(* LS Electric XG5000 project: Test_260202 *)
(* PLC LSPLC *)
(* module base 0 slot 0: FEnet:XGL-EFMT(B) (Fast Ethernet 통신 모듈, 전기 Master) *)
(* module base 0 slot 1: 입력 모듈:XGI-D21A (DC 24V 입력, 8점 (전류소스/싱크입력)) *)
(* module base 0 slot 2: 출력 모듈:XGQ-RY1A (릴레이 출력, 8점 (2A용, 단독 COM.)) *)

(* Comments on direct variables
%MX0	Emitter 0 (Emit)
%MX1	E_Belt 0
%MX2	Emitter 1 (Emit)
%MX3	E_Belt 1
%MX4	Emitter 2 (Emit)
%MX5	E_Belt 2
%MX6	Emitter 3 (Emit)
%MX7	E_Belt 3
%MX8	Emitter 4 (Emit)
%MX9	E_Belt 4
%MX10	Emitter 5 (Emit)
%MX11	E_Belt 5
%MX12	P_Belt00
%MX13	Sensor P_Belt00_E
%MX14	P_Belt0
%MX15	Sensor P_Belt0_E
%MX16	Sensor P_Belt0_S
%MX17	P_Belt1
%MX18	Sensor P_Belt1_E
%MX19	Sensor P_Belt1_S
%MX20	P_Belt2
%MX21	Sensor P_Belt2_E
%MX22	Sensor P_Belt2_S
%MX23	P_Belt3
%MX24	Sensor P_Belt3_E
%MX25	Sensor P_Belt3_S
%MX26	P_Belt4
%MX27	Sensor P_Belt4_E
%MX28	Sensor P_Belt4_S
%MX29	P_Belt5
%MX30	Sensor P_Belt5_E
%MX31	Sensor P_Belt5_S
%MX32	P_Belt6
%MX33	Sensor P_Belt6_S
%MX34	Sensor P_Belt6_E
%MX35	CC_Belt0
%MX36	Sensor CC_Belt0
%MX37	Sensor CC_Belt1
%MX38	Sensor CC_Belt2
%MX39	Pusher 0
%MX40	Pusher 1
%MX41	Pusher 2
%MX42	Pusher 3
%MX43	Pusher 4
%MX44	CG_Belt1
%MX45	CG_Belt2
%MX46	CG_Curved Belt0
%MX47	CGD_Belt0
%MX48	CGD_Belt1
%MX49	CGD_Belt2
%MX50	CGD_Belt3
%MX51	Sensor Divide_G
%MX52	Sensor Error0
%MX53	Sensor_Count_Green
%MX54	CB_Belt1
%MX55	CB_Curved Belt0
%MX56	CBD_Belt0
%MX57	CBD_Belt1
%MX58	CBD_Belt2
%MX59	CBD_Belt3
%MX60	CBD_Belt4
%MX61	Pusher 5
%MX62	Pusher 6
%MX63	Sensor Divide_B
%MX64	Sensor Error1
%MX65	Sensor_Count_Blue
%MX66	CM_Belt1
%MX67	CM_Curved Belt0
%MX68	CMD_Belt0
%MX69	CMD_Belt1
%MX70	CMD_Belt2
%MX71	CMD_Belt3
%MX72	CMD_Belt4
%MX73	Pusher 7
%MX74	Pusher 8
%MX75	Sensor Divide_M
%MX76	Sensor Error2
%MX77	Sensor_Count_Metal
%MX100	A_Belt blue Conveyor
%MX101	A_Entry conveyor
%MX102	A_Start Entry Conveyor
%MX103	A_Item at entry
%MX104	A_Box at place
%MX105	A_Box Pass
%MX106	A_Box exit Conveyor
%MX107	A_Chain Transfer1 
%MX108	A_Chain Transfer2
%MX109	A_Transfer1 (Left)
%MX110	A_Transfer2 (Left)
%MX111	A_Direction Change
%MX112	A_Box entry to ware
%MX113	A_Box entry warehouse
%MX114	A_Box Check
%MX115	WA_Entry conveyor
%MX116	B_Belt Green Conveyor
%MX117	B_Entry conveyor
%MX118	B_Start Entry Conveyor
%MX119	B_Item at entry
%MX120	B_Box at place
%MX121	B_Box Pass
%MX122	B_Box exit Conveyor1
%MX123	B_Go
%MX124	B_Box arrive
%MX125	B_return
%MX126	B_Box Pass2
%MX127	B_Box exit Conveyor2
%MX128	B_Chain Transfer1 
%MX129	B_Chain Transfer2
%MX130	B_Direction Change
%MX131	B_Transfer1 (Right)
%MX132	B_Transfer2 (Right)
%MX133	B_Box entry to ware
%MX134	B_Box entry warehouse
%MX135	B_Box Check
%MX136	WB_Entry conveyor
%MX137	C_Belt Gray Conveyor
%MX138	C_Start Entry Conveyor
%MX139	C_Entry conveyor
%MX140	C_Item at entry
%MX141	C_Exit Conveyor
%MX142	C_Box Pass
%MX143	C_Box Pass2
%MX144	C_Exit Conveyor
%MX145	C_Chain Transfer1 
%MX146	C_Chain Transfer2
%MX147	C_Direction Change
%MX148	C_Transfer1 (Right)
%MX149	C_Transfer2 (Right)
%MX150	C_Box entry to ware
%MX151	C_Box entry warehouse
%MX152	WC_Entry conveyor
%MX500	Out_Conv_1_In_Sensor
%MX501	Out_Conv_1_Out_Sensor
%MX502	Out_Conv_2_In_Sensor
%MX503	Out_Conv_2_Out_Sensor
%MX504	Out_Conv_3_In_Sensor
%MX505	Out_Conv_3_Out_Sensor
%MX506	Out_Conv_4_In_Sensor
%MX507	Out_Conv_4_Out_Sensor
%MX508	Out_Conv_Line1-1_In_Sensor
%MX509	Out_Conv_Line1-1_Out_Sensor
%MX510	Out_Conv_Line1-2_In_Sensor
%MX511	Out_Conv_Line1-2_Out_Sensor
%MX512	Out_Conv_Line1-3_In_Sensor
%MX513	Out_Conv_Line1-3_Out_Sensor
%MX514	Out_Conv_Line1-4_In_Sensor
%MX515	Out_Conv_Line1-4_Out_Sensor
%MX516	Out_Conv_Line2-1_In_Sensor
%MX517	Out_Conv_Line2-1_Out_Sensor
%MX518	Out_Conv_Line2-2_In_Sensor
%MX519	Out_Conv_Line2-2_Out_Sensor
%MX520	Out_Conv_Line2-3_In_Sensor
%MX521	Out_Conv_Line2-3_Out_Sensor
%MX522	Out_Conv_Line2-4_In_Sensor
%MX523	Out_Conv_Line2-4_Out_Sensor
%MX524	Out_Conv_Line2-5_In_Sensor
%MX525	Out_Conv_Line2-5_Out_Sensor
%MX526	Out_Conv_Line3-1_In_Sensor
%MX527	Out_Conv_Line3-1_Out_Sensor
%MX528	Out_Conv_Line3-2_In_Sensor
%MX529	Out_Conv_Line3-2_Out_Sensor
%MX530	Out_Conv_Line3-3_In_Sensor
%MX531	Out_Conv_Line3-3_Out_Sensor
%MX532	Out_Conv_Line3-4_In_Sensor
%MX533	Out_Conv_Line3-4_Out_Sensor
%MX1000	Start_Button 0
%MX1001	Stop_Button 0
%MX1002	Emergency Stop 0
%MX1003	Machining Center 0 (Is Busy)
%MX1004	Machining Center 0 (Has Error)
%MX1005	Start_Button 1
%MX1006	Stop_Button 1
%MX1007	Emergency Stop 1
%MX1008	Machining Center 1 (Is Busy)
%MX1009	Machining Center 1 (Has Error)
%MX1010	Start_Button 2
%MX1011	Stop_Button 2
%MX1012	Emergency Stop 2
%MX1013	Machining Center 2 (Is Busy)
%MX1014	Machining Center 2 (Has Error)
%MX1015	Start_Button 3
%MX1016	Stop_Button 3
%MX1017	Emergency Stop 3
%MX1018	Machining Center 3 (Is Busy)
%MX1019	Machining Center 3 (Has Error)
%MX1020	C_Start Button 0
%MX1021	C_Stop Button 0
%MX1022	C_Emergency Stop 0
%MX1023	Vision Sensor 0
%MX1024	Vision Sensor 1
%MX1025	Vision Sensor 2
%MX1026	Vision Sensor 3
%MX1027	Vision Sensor 4
%MX1028	Vision Sensor 5
%MX1029	Pusher 0 (Front Limit)
%MX1030	Pusher 1 (Front Limit)
%MX1031	Pusher 2 (Front Limit)
%MX1032	Vision Sensor 6
%MX1033	Vision Sensor 7
%MX1034	Vision Sensor 8
%MX1035	Vision Sensor 9
%MX1036	Vision Sensor 10
%MX1037	Vision Sensor 11
%MX1038	Pusher 3 (Front Limit)
%MX1039	Pusher 4 (Front Limit)
%MX1040	Pusher 5 (Front Limit)
%MX1041	Pusher 6 (Front Limit)
%MX1042	Pusher 7 (Front Limit)
%MX1043	Pusher 8 (Front Limit)
%MX1044	Diffuse Sensor 4
%MX1045	Diffuse Sensor 5
%MX1046	Right Positioner 0 (Clamped)
%MX1047	Right Positioner 1 (Clamped)
%MX1048	Two-Axis Pick & Place 0 (Detected)
%MX1049	Two-Axis Pick & Place 0 (Moving X)
%MX1050	Two-Axis Pick & Place 0 (Moving Z)
%MX1051	Clamp_Sensor 0
%MX1052	Clamp_Sensor 1
%MX1053	Combine Sensor 0
%MX1054	RaiseDown_Sensor 0
%MX1055	Start_Button 4
%MX1056	Stop_Button 4
%MX1057	Emergency Stop 4
%MX1058	Machining Center 4 (Is Busy)
%MX1059	Machining Center 4 (Has Error)
%MX1060	Start_Button 5
%MX1061	Stop_Button 5
%MX1062	Emergency Stop 5
%MX1063	Machining Center 5 (Is Busy)
%MX1064	Machining Center 5 (Has Error)
%MX1065	Diffuse Sensor 6
%MX1066	Diffuse Sensor 7
%MX1067	Right Positioner 2 (Clamped)
%MX1068	Right Positioner 3 (Clamped)
%MX1069	Two-Axis Pick & Place 1 (Detected)
%MX1070	Two-Axis Pick & Place 1 (Moving X)
%MX1071	Two-Axis Pick & Place 1 (Moving Z)
%MX1072	Clamp_Sensor 2
%MX1073	Clamp_Sensor 3
%MX1074	Combine Sensor 1
%MX1075	RaiseDown_Sensor 1
%MX1076	Diffuse Sensor 8
%MX1077	Diffuse Sensor 9
%MX1078	Right Positioner 4 (Clamped)
%MX1079	Right Positioner 5 (Clamped)
%MX1080	Two-Axis Pick & Place 2 (Detected)
%MX1081	Two-Axis Pick & Place 2 (Moving X)
%MX1082	Two-Axis Pick & Place 2 (Moving Z)
%MX1083	Clamp_Sensor 4
%MX1084	Clamp_Sensor 5
%MX1085	Combine Sensor 2
%MX1086	RaiseDown_Sensor 2
%MX1087	Sensor Error0
%MX1088	Sensor Error1
%MX1089	Sensor Error2
%MX1090	Sensor_Count_Green
%MX1091	Sensor_Count_Blue
%MX1092	Sensor_Count_Metal
%MX1093	Reset Button_Green
%MX1094	Reset Button_Blue
%MX1095	Reset Button_Metal
%MX1101	Sensor CC_Belt0
%MX1102	Sensor CC_Belt1
%MX1103	Sensor CC_Belt2
%MX1104	Sensor Divide_G
%MX1105	Sensor Divide_B
%MX1106	Sensor Divide_M
%MX1110	Sensor P_Belt00_E
%MX1111	Sensor P_Belt0_E
%MX1112	Sensor P_Belt0_S
%MX1113	Sensor P_Belt1_E
%MX1114	Sensor P_Belt1_S
%MX1115	Sensor P_Belt2_E
%MX1116	Sensor P_Belt2_S
%MX1117	Sensor P_Belt3_E
%MX1118	Sensor P_Belt3_S
%MX1119	Sensor P_Belt4_E
%MX1120	Sensor P_Belt4_S
%MX1121	Sensor P_Belt5_E
%MX1122	Sensor P_Belt5_S
%MX1123	Sensor P_Belt6_E
%MX1124	Sensor P_Belt6_S
%MX2000	Start Button 0 (Light)
%MX2001	Stop Button 0 (Light)
%MX2002	Emitter 0 (Emit)
%MX2003	E_Belt 0
%MX2004	Machining Center 0 (Start)
%MX2005	Machining Center 0 (Stop)
%MX2006	Start Button 1 (Light)
%MX2007	Stop Button 1 (Light)
%MX2008	Emitter 1 (Emit)
%MX2009	E_Belt 1
%MX2010	Machining Center 1 (Start)
%MX2011	Machining Center 1 (Stop)
%MX2012	Start Button 2 (Light)
%MX2013	Stop Button 2 (Light)
%MX2014	Emitter 2 (Emit)
%MX2015	E_Belt 2
%MX2016	Machining Center 2 (Start)
%MX2017	Machining Center 2 (Stop)
%MX2018	Start Button 3 (Light)
%MX2019	Stop Button 3 (Light)
%MX2020	Emitter 3 (Emit)
%MX2021	E_Belt 3
%MX2022	Machining Center 3 (Start)
%MX2023	Machining Center 3 (Stop)
%MX2024	P_Belt0
%MX2025	P_Belt1
%MX2026	P_Belt2
%MX2027	P_Belt3
%MX2028	P_Curved Belt0
%MX2029	CC_Belt0
%MX2030	CG_Belt1
%MX2031	CG_Belt2
%MX2032	CG_Curved Belt0
%MX2033	CGD_Belt0
%MX2034	CGD_Belt1
%MX2035	CGD_Belt2
%MX2036	CGD_Belt3
%MX2037	CB_Belt1
%MX2038	CB_Curved Belt0
%MX2039	CBD_Belt0
%MX2040	CBD_Belt1
%MX2041	CBD_Belt2
%MX2042	CBD_Belt3
%MX2043	CBD_Belt4
%MX2044	CM_Belt1
%MX2045	CM_Curved Belt0
%MX2046	CMD_Belt0
%MX2047	CMD_Belt1
%MX2048	CMD_Belt2
%MX2049	CMD_Belt3
%MX2050	CMD_Belt4
%MX2051	C_Start Button 0(Light)
%MX2052	C_Stop Button 0 (Light)
%MX2053	Pusher 0
%MX2054	Pusher 1
%MX2055	Pusher 2
%MX2056	Pusher 3
%MX2057	Pusher 4
%MX2058	Pusher 5
%MX2059	Pusher 6
%MX2060	Pusher 7
%MX2061	Pusher 8
%MX2062	Right Positioner 0 (Clamp)
%MX2063	Right Positioner 0 (Raise)
%MX2064	Right Positioner 1 (Clamp)
%MX2065	Two-Axis Pick & Place 0 X
%MX2066	Two-Axis Pick & Place 0 Z
%MX2067	Two-Axis Pick & Place 0 (Grab)
%MX2068	Start Button 4 (Light)
%MX2069	Stop Button 4 (Light)
%MX2070	Emitter 4 (Emit)
%MX2071	E_Belt 4
%MX2072	Machining Center 4 (Start)
%MX2073	Machining Center 4 (Stop)
%MX2074	Start Button 5 (Light)
%MX2075	Stop Button 5 (Light)
%MX2076	Emitter 5 (Emit)
%MX2077	E_Belt 5
%MX2078	Machining Center 5 (Start)
%MX2079	Machining Center 5 (Stop)
%MX2080	P_Belt4
%MX2081	P_Belt5
%MX2082	P_Belt6
%MX2083	Right Positioner 2 (Clamp)
%MX2084	Right Positioner 2 (Raise)
%MX2085	Right Positioner 3 (Clamp)
%MX2086	Two-Axis Pick & Place 1 X
%MX2087	Two-Axis Pick & Place 1 Z
%MX2088	Two-Axis Pick & Place 1 (Grab)
%MX2089	Right Positioner 4 (Clamp)
%MX2090	Right Positioner 4 (Raise)
%MX2091	Right Positioner 5 (Clamp)
%MX2092	Two-Axis Pick & Place 2 X
%MX2093	Two-Axis Pick & Place 2 Z
%MX2094	Two-Axis Pick & Place 2 (Grab)
%MX2095	Right Positioner 1 (Raise)
%MX2096	Right Positioner 3 (Raise)
%MX2097	Right Positioner 5 (Raise)
%MX2098	P_Belt00
%MX2099	Reset Button_Green (Light)
%MX2100	Reset Button_Blue (Light)
%MX2101	Reset Button_Metal (Light)
%MX3000	스타트버튼유지0
%MX3001	생산기계유지0
%MX3002	스탑버튼유지0
%MX3003	스타트버튼유지1
%MX3004	생산기계유지1
%MX3005	스탑버튼유지1
%MX3006	스타트버튼유지2
%MX3007	생산기계유지2
%MX3008	스탑버튼유지2
%MX3009	스타트버튼유지3
%MX3010	생산기계유지3
%MX3011	스탑버튼유지3
%MX3012	C_Start유지
%MX3013	푸쉬0유지
%MX3014	푸쉬1유지
%MX3015	푸쉬2유지
%MX3016	푸쉬3유지
%MX3017	푸쉬4유지
%MX3018	푸쉬5유지
%MX3019	푸쉬6유지
%MX3020	푸쉬7유지
%MX3021	푸쉬8유지
%MX3022	클램프0유지
%MX3023	클램프1유지
%MX3024	Grab유지
%MX3025	Move 0 Z
%MX3026	Move 0 X
%MX3027	Move 1 Z
%MX3028	Grab해제
%MX3029	Clamp_Raise
%MX3030	스타트버튼유지4
%MX3031	생산기계유지4
%MX3032	스탑버튼유지4
%MX3033	스타트버튼유지5
%MX3034	생산기계유지5
%MX3035	스탑버튼유지5
%MX3036	클램프2유지
%MX3037	클램프3유지
%MX3038	Grab유지
%MX3039	Move 0 Z
%MX3040	Move 0 X
%MX3041	Move 1 Z
%MX3042	Grab해제
%MX3043	Clamp_Raise
%MX3044	클램프4유지
%MX3045	클램프5유지
%MX3046	Grab유지
%MX3047	Move 0 Z
%MX3048	Move 0 X
%MX3049	Move 1 Z
%MX3050	Grab해제
%MX3051	Clamp_Raise
%MX3103	OpenCV_데이터값Read(초록)
%MX3104	OpenCV_데이터값Read(파랑)
%MX3105	OpenCV_데이터값Read(메탈)
%MX3106	OpenCV_데이터값Read(뚜껑)
%MX3107	ReadData_초록
%MX3108	ReadData_파랑
%MX3109	ReadData_메탈
%MX3110	ReadData_뚜껑
%MX3200	Sensor CC_Belt1 자기유지 회로
%MX3201	Sensor Divide_G 자기유지 회로
%MX3202	Sensor Divide_B 자기유지 회로
%MX3203	Sensor Divide_M 자기유지 회로
%MX4000	A_Start
%MX4001	A_Stop
%MX4002	A_Item at entry
%MX4003	A_Box at exit
%MX4004	A_Start Entry Conveyor
%MX4005	A_Auto
%MX4006	A_Manual
%MX4007	A_Item detected
%MX4008	A_Item at exit
%MX4009	A_Moving X
%MX4010	A_Moving Z
%MX4011	A_Box at place
%MX4012	A_Box Pass2
%MX4013	A_Box Pass
%MX4014	A_Direction Change
%MX4015	A_Box Check
%MX4016	A_Box entry to ware
%MX4017	A_Box Emergency stop
%MX4030	B_Start
%MX4031	B_Stop
%MX4032	B_Item at entry
%MX4033	B_Box at exit
%MX4034	B_Start Entry Conveyor
%MX4035	B_Auto
%MX4036	B_Manual
%MX4037	B_Item detected
%MX4038	B_Item at exit
%MX4039	B_Moving X
%MX4040	B_Moving Z
%MX4041	B_Box at place
%MX4042	B_Box Pass2
%MX4043	B_Box Pass
%MX4044	B_Direction Change
%MX4045	B_Box Check
%MX4046	B_Box entry to ware
%MX4047	B_Turn entry
%MX4048	B_Box arrive
%MX4049	B_Go
%MX4050	B_return
%MX4051	B_Box Emergency stop
%MX4060	C_Start
%MX4061	C_Stop
%MX4062	C_Item at entry
%MX4063	C_Box at exit
%MX4064	C_Start Entry Conveyor
%MX4065	C_Auto
%MX4066	C_Manual
%MX4067	C_Item detected
%MX4068	C_Item at exit
%MX4069	C_Moving X
%MX4070	C_Moving Z
%MX4071	C_Box at place
%MX4072	C_Box Pass2
%MX4073	C_Box Pass
%MX4074	C_Direction Change
%MX4075	C_Box Check
%MX4076	C_Box entry to ware
%MX4077	C_Box Emergency stop
%MX4100	WA_Start Button
%MX4101	WA_Stop Button
%MX4102	WA_Reset Button
%MX4103	WA_Auto
%MX4104	WA_Manual
%MX4105	WA_emergency stop
%MX4106	WA_Diffuse Sensor
%MX4110	WB_Start Button
%MX4111	WB_Stop Button
%MX4112	WB_Reset Button
%MX4113	WB_Auto
%MX4114	WB_Manual
%MX4115	WB_emergency stop
%MX4116	WB_Diffuse Sensor
%MX4120	WC_Start Button
%MX4121	WC_Stop Button
%MX4122	WC_Reset Button
%MX4123	WC_Auto
%MX4124	WC_Manual
%MX4125	WC_emergency stop
%MX4126	WC_Diffuse Sensor
%MX4130	All_Start
%MX4131	All_Stop
%MX4132	All_Emergency Stop
%MX4133	All_Manual
%MX4134	All_Auto
%MX5000	A_Belt blue Conveyor
%MX5001	A_Entry conveyor
%MX5002	A_Move Z
%MX5003	A_Grab
%MX5004	A_Exit Conveyor
%MX5005	A_Move X
%MX5006	A_Light 1 (Green)
%MX5007	A_Light 1 (Yellow)
%MX5008	A_Light 2 (Green)
%MX5009	A_Light 2 (Yellow)
%MX5010	A_Light 1 (Red)
%MX5011	A_Light 2 (Red)
%MX5012	A_Box exit Conveyor
%MX5013	A_Chain Transfer1 
%MX5014	A_Chain Transfer2
%MX5015	A_Transfer1 (Left)
%MX5016	A_Transfer2 (Left)
%MX5017	A_Box entry warehouse
%MX5018	A_Box emitter
%MX5030	B_Belt Green Conveyor
%MX5031	B_Entry conveyor
%MX5032	B_Move Z
%MX5033	B_Grab
%MX5034	B_Exit Conveyor
%MX5035	B_Move X
%MX5036	B_Light 1 (Green)
%MX5037	B_Light 1 (Yellow)
%MX5038	B_Light 2 (Green)
%MX5039	B_Light 2 (Yellow)
%MX5040	B_Light 1 (Red)
%MX5041	B_Light 2 (Red)
%MX5042	B_Box exit Conveyor1
%MX5043	B_Box exit Conveyor2
%MX5044	B_Chain Transfer1 
%MX5045	B_Chain Transfer2
%MX5046	B_Transfer1 (Right)
%MX5047	B_Transfer2 (Right)
%MX5048	B_Box entry warehouse
%MX5049	B_Box emitter
%MX5050	B_Turntable Roll (+)
%MX5051	B_Turntable Roll (-)
%MX5052	B_Turntable Turn
%MX5060	C_Belt Gray Conveyor
%MX5061	C_Entry conveyor
%MX5062	C_Move Z
%MX5063	C_Grab
%MX5064	C_Exit Conveyor
%MX5065	C_Move X
%MX5066	C_Light 1 (Green)
%MX5067	C_Light 1 (Yellow)
%MX5068	C_Light 2 (Green)
%MX5069	C_Light 2 (Yellow)
%MX5070	C_Light 1 (Red)
%MX5071	C_Light 2 (Red)
%MX5072	C_Box exit Conveyor
%MX5073	C_Chain Transfer1 
%MX5074	C_Chain Transfer2
%MX5075	C_Transfer1 (Right)
%MX5076	C_Transfer2 (Right)
%MX5077	C_Box entry warehouse
%MX5078	C_Box emitter
%MX5100	WA_Load Conveyor
%MX5101	WA_forks left
%MX5102	WA_forks right
%MX5103	WA_Lift
%MX5104	WA_Start Light
%MX5105	WA_Stop Light
%MX5106	WA_Entry conveyor
%MX5107	WA_Reset Light
%MX5108	WA_Stopper
%MX5110	WB_Load Conveyor
%MX5111	WB_forks left
%MX5112	WB_forks right
%MX5113	WB_Lift
%MX5114	WB_Start Light
%MX5115	WB_Stop Light
%MX5116	WB_Entry conveyor
%MX5117	WB_Reset Light
%MX5118	WB_Stopper
%MX5120	WC_Load Conveyor
%MX5121	WC_forks left
%MX5122	WC_forks right
%MX5123	WC_Lift
%MX5124	WC_Start Light
%MX5125	WC_Stop Light
%MX5126	WC_Entry conveyor
%MX5127	WC_Reset Light
%MX5128	WC_Stopper
%MX6000	A_Blue Line Run
%MX6001	A_Stop
%MX6002	A_Entry conveyor
%MX6003	A_Started
%MX6004	A_Move Z 1
%MX6005	A_Move Z 2
%MX6006	A_Grab
%MX6007	A_Move X 1
%MX6008	A_Exit conveyor
%MX6009	A_Box exit 1
%MX6010	A_Box exit 2
%MX6011	A_Box exit 3
%MX6012	A_Box exit 4
%MX6030	B_Green Line Run
%MX6031	B_Stop
%MX6032	B_Entry conveyor
%MX6033	B_Started
%MX6034	B_Move Z 1
%MX6035	B_Move Z 2
%MX6036	B_Grab
%MX6037	B_Move X 1
%MX6038	B_Exit conveyor
%MX6039	B_Box exit 1
%MX6040	B_Box exit 2
%MX6041	B_Box exit 3
%MX6042	B_Box exit 4
%MX6043	B_Turntable Roll (+)
%MX6044	B_Turntable Roll (-)
%MX6045	B_Turntable Turn
%MX6046	B_Box exit Conveyor2
%MX6060	C_Gray Line Run
%MX6061	C_Stop
%MX6062	C_Entry conveyor
%MX6063	C_Started
%MX6064	C_Move Z 1
%MX6065	C_Move Z 2
%MX6066	C_Grab
%MX6067	C_Move X 1
%MX6068	C_Exit conveyor
%MX6069	C_Box exit 1
%MX6070	C_Box exit 2
%MX6071	C_Box exit 3
%MX6072	C_Box exit 4
%MX6100	WA_Run_System
%MX6110	WB_Run_System
%MX6120	WC_Run_System
%MX6130	All_Run_System
%MX6131	All_Stop_System
*)

PROGRAM NewProgram (* task: 스캔 프로그램 *)

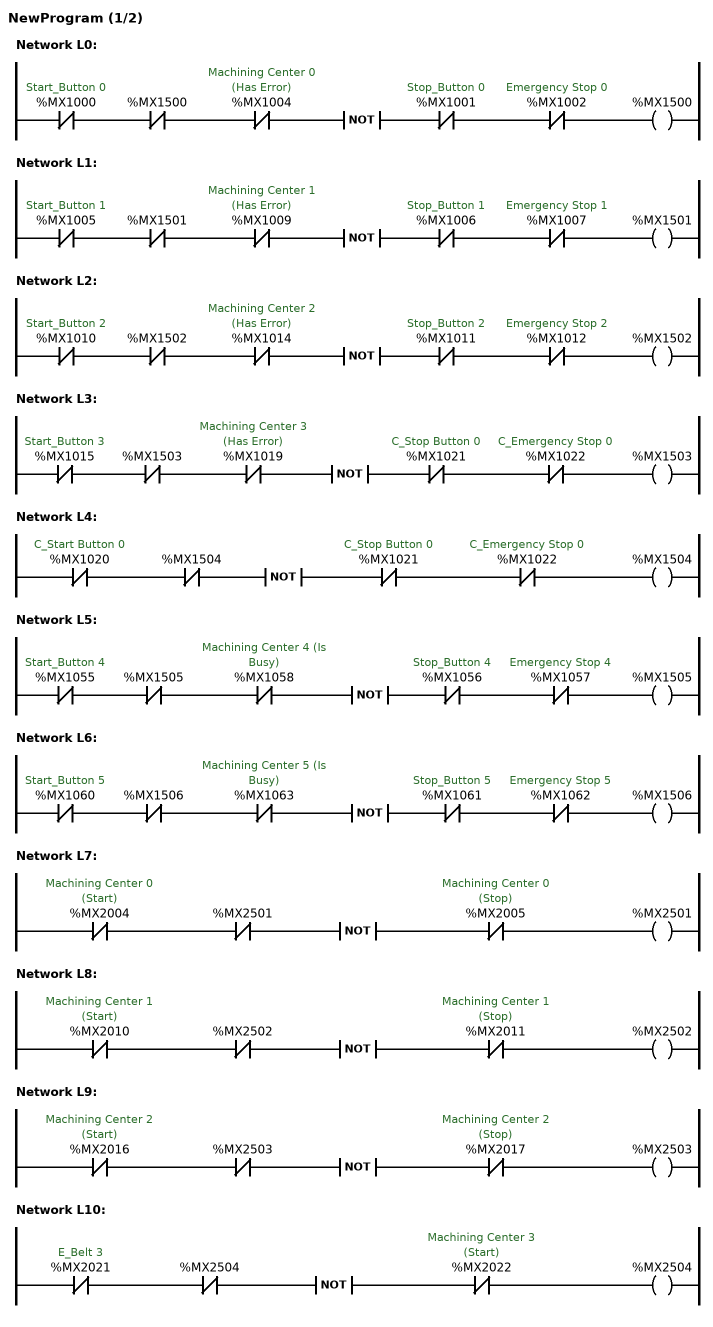
(* Rung L0 *)
%MX1500 := NOT (NOT %MX1000 AND NOT %MX1500 AND NOT %MX1004) AND NOT %MX1001 AND NOT %MX1002;
(* Rung L1 *)
%MX1501 := NOT (NOT %MX1005 AND NOT %MX1501 AND NOT %MX1009) AND NOT %MX1006 AND NOT %MX1007;
(* Rung L2 *)
%MX1502 := NOT (NOT %MX1010 AND NOT %MX1502 AND NOT %MX1014) AND NOT %MX1011 AND NOT %MX1012;
(* Rung L3 *)
%MX1503 := NOT (NOT %MX1015 AND NOT %MX1503 AND NOT %MX1019) AND NOT %MX1021 AND NOT %MX1022;
(* Rung L4 *)
%MX1504 := NOT (NOT %MX1020 AND NOT %MX1504) AND NOT %MX1021 AND NOT %MX1022;
(* Rung L5 *)
%MX1505 := NOT (NOT %MX1055 AND NOT %MX1505 AND NOT %MX1058) AND NOT %MX1056 AND NOT %MX1057;
(* Rung L6 *)
%MX1506 := NOT (NOT %MX1060 AND NOT %MX1506 AND NOT %MX1063) AND NOT %MX1061 AND NOT %MX1062;
(* Rung L7 *)
%MX2501 := NOT (NOT %MX2004 AND NOT %MX2501) AND NOT %MX2005;
(* Rung L8 *)
%MX2502 := NOT (NOT %MX2010 AND NOT %MX2502) AND NOT %MX2011;
(* Rung L9 *)
%MX2503 := NOT (NOT %MX2016 AND NOT %MX2503) AND NOT %MX2017;
(* Rung L10 *)
%MX2504 := NOT (NOT %MX2021 AND NOT %MX2504) AND NOT %MX2022;

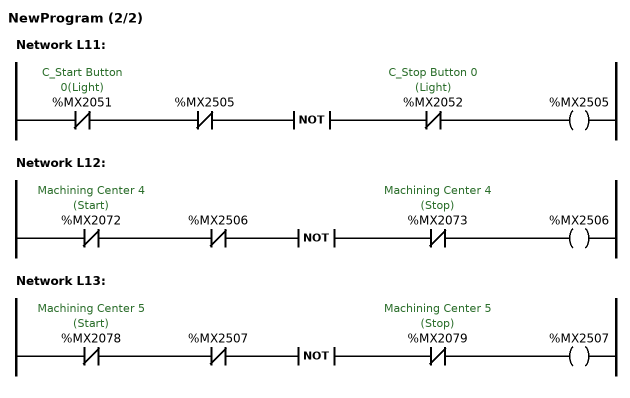
(* Rung L11 *)
%MX2505 := NOT (NOT %MX2051 AND NOT %MX2505) AND NOT %MX2052;
(* Rung L12 *)
%MX2506 := NOT (NOT %MX2072 AND NOT %MX2506) AND NOT %MX2073;
(* Rung L13 *)
%MX2507 := NOT (NOT %MX2078 AND NOT %MX2507) AND NOT %MX2079;
END_PROGRAM

PROGRAM Communication (* task: 스캔 프로그램 *)
VAR
    Camera1 : TON;
    Camera2 : TON;
END_VAR

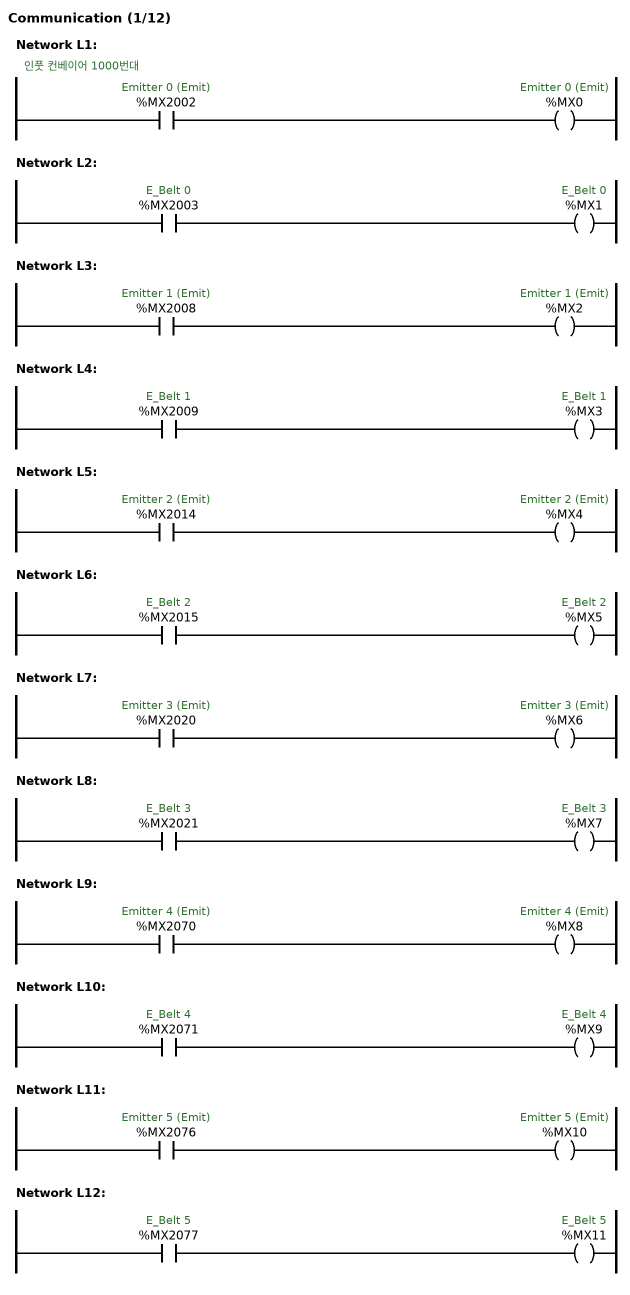
(* 인풋 컨베이어 1000번대 *)
(* Rung L1 *)
%MX0 := %MX2002;
(* Rung L2 *)
%MX1 := %MX2003;
(* Rung L3 *)
%MX2 := %MX2008;
(* Rung L4 *)
%MX3 := %MX2009;
(* Rung L5 *)
%MX4 := %MX2014;
(* Rung L6 *)
%MX5 := %MX2015;
(* Rung L7 *)
%MX6 := %MX2020;
(* Rung L8 *)
%MX7 := %MX2021;
(* Rung L9 *)
%MX8 := %MX2070;
(* Rung L10 *)
%MX9 := %MX2071;
(* Rung L11 *)
%MX10 := %MX2076;
(* Rung L12 *)
%MX11 := %MX2077;

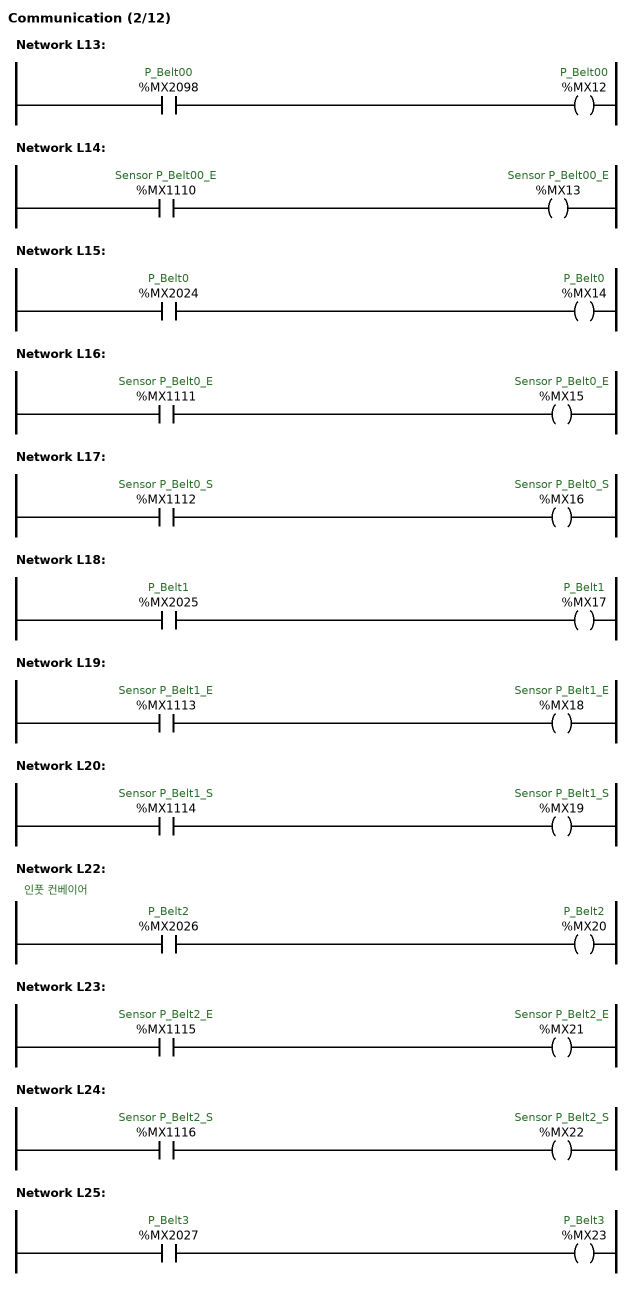
(* Rung L13 *)
%MX12 := %MX2098;
(* Rung L14 *)
%MX13 := %MX1110;
(* Rung L15 *)
%MX14 := %MX2024;
(* Rung L16 *)
%MX15 := %MX1111;
(* Rung L17 *)
%MX16 := %MX1112;
(* Rung L18 *)
%MX17 := %MX2025;
(* Rung L19 *)
%MX18 := %MX1113;
(* Rung L20 *)
%MX19 := %MX1114;
(* 인풋 컨베이어 *)
(* Rung L22 *)
%MX20 := %MX2026;
(* Rung L23 *)
%MX21 := %MX1115;
(* Rung L24 *)
%MX22 := %MX1116;
(* Rung L25 *)
%MX23 := %MX2027;

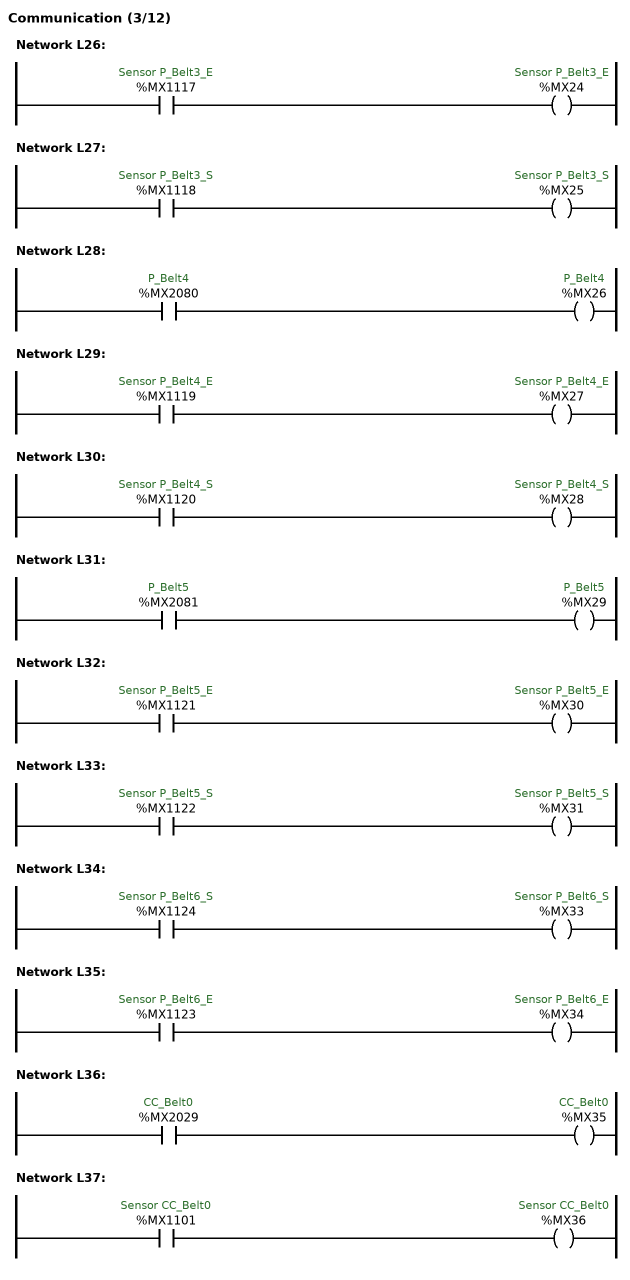
(* Rung L26 *)
%MX24 := %MX1117;
(* Rung L27 *)
%MX25 := %MX1118;
(* Rung L28 *)
%MX26 := %MX2080;
(* Rung L29 *)
%MX27 := %MX1119;
(* Rung L30 *)
%MX28 := %MX1120;
(* Rung L31 *)
%MX29 := %MX2081;
(* Rung L32 *)
%MX30 := %MX1121;
(* Rung L33 *)
%MX31 := %MX1122;
(* Rung L34 *)
%MX33 := %MX1124;
(* Rung L35 *)
%MX34 := %MX1123;
(* Rung L36 *)
%MX35 := %MX2029;
(* Rung L37 *)
%MX36 := %MX1101;

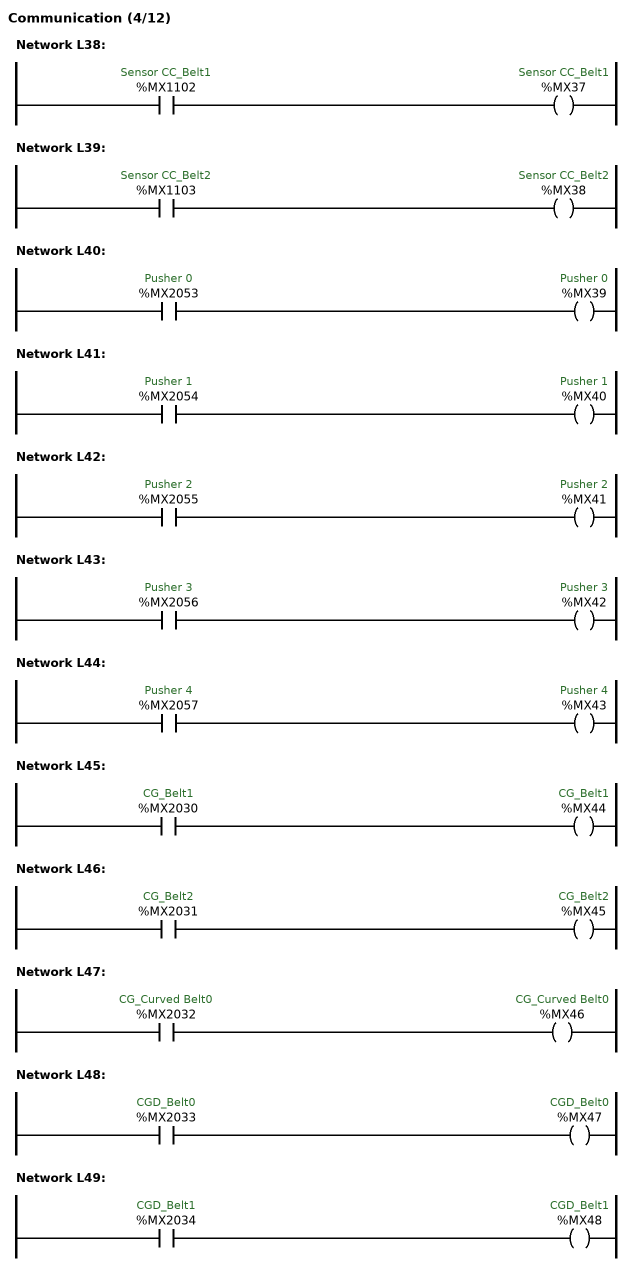
(* Rung L38 *)
%MX37 := %MX1102;
(* Rung L39 *)
%MX38 := %MX1103;
(* Rung L40 *)
%MX39 := %MX2053;
(* Rung L41 *)
%MX40 := %MX2054;
(* Rung L42 *)
%MX41 := %MX2055;
(* Rung L43 *)
%MX42 := %MX2056;
(* Rung L44 *)
%MX43 := %MX2057;
(* Rung L45 *)
%MX44 := %MX2030;
(* Rung L46 *)
%MX45 := %MX2031;
(* Rung L47 *)
%MX46 := %MX2032;
(* Rung L48 *)
%MX47 := %MX2033;
(* Rung L49 *)
%MX48 := %MX2034;

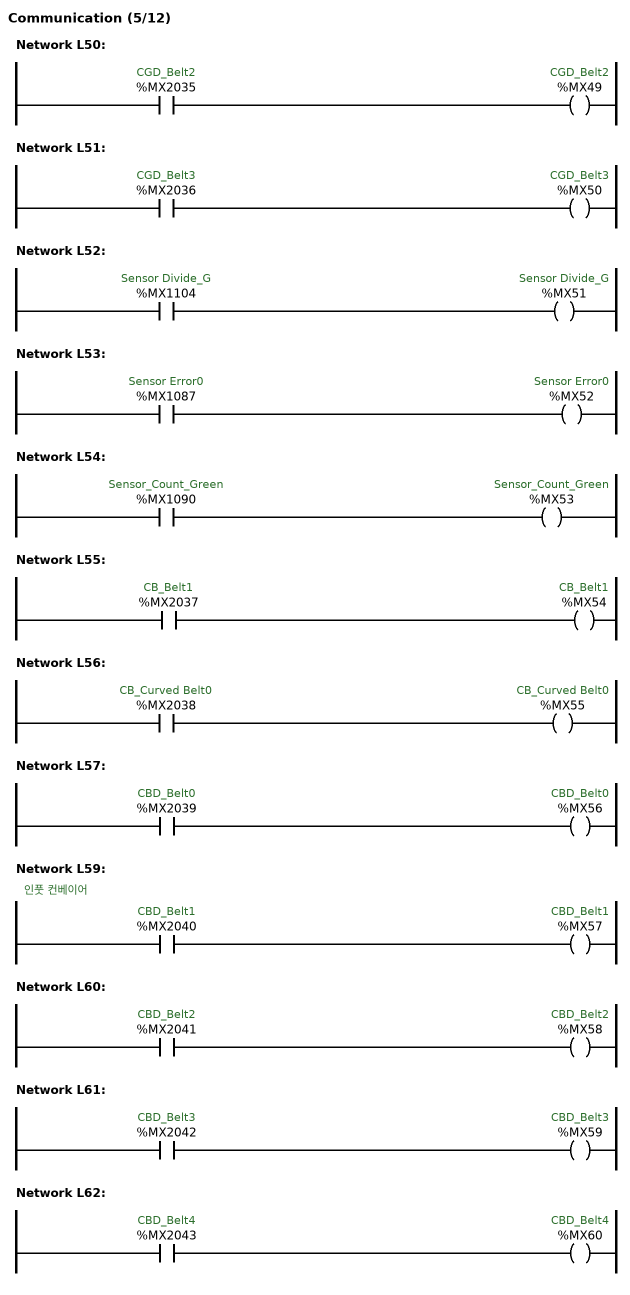
(* Rung L50 *)
%MX49 := %MX2035;
(* Rung L51 *)
%MX50 := %MX2036;
(* Rung L52 *)
%MX51 := %MX1104;
(* Rung L53 *)
%MX52 := %MX1087;
(* Rung L54 *)
%MX53 := %MX1090;
(* Rung L55 *)
%MX54 := %MX2037;
(* Rung L56 *)
%MX55 := %MX2038;
(* Rung L57 *)
%MX56 := %MX2039;
(* 인풋 컨베이어 *)
(* Rung L59 *)
%MX57 := %MX2040;
(* Rung L60 *)
%MX58 := %MX2041;
(* Rung L61 *)
%MX59 := %MX2042;
(* Rung L62 *)
%MX60 := %MX2043;

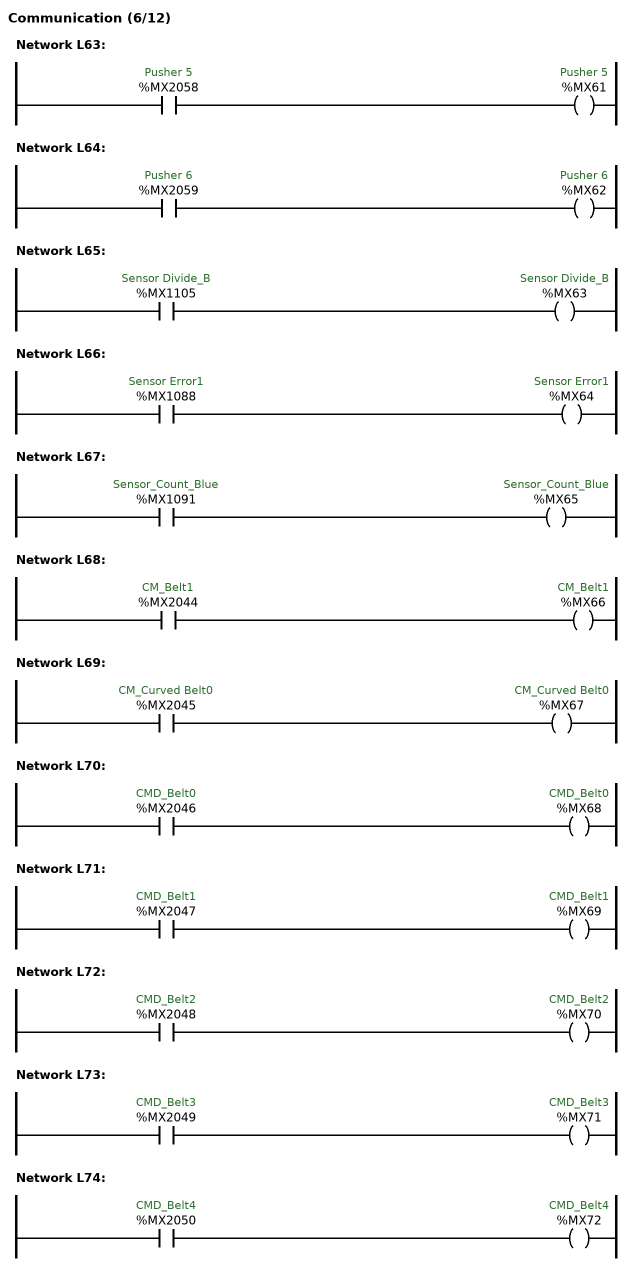
(* Rung L63 *)
%MX61 := %MX2058;
(* Rung L64 *)
%MX62 := %MX2059;
(* Rung L65 *)
%MX63 := %MX1105;
(* Rung L66 *)
%MX64 := %MX1088;
(* Rung L67 *)
%MX65 := %MX1091;
(* Rung L68 *)
%MX66 := %MX2044;
(* Rung L69 *)
%MX67 := %MX2045;
(* Rung L70 *)
%MX68 := %MX2046;
(* Rung L71 *)
%MX69 := %MX2047;
(* Rung L72 *)
%MX70 := %MX2048;
(* Rung L73 *)
%MX71 := %MX2049;
(* Rung L74 *)
%MX72 := %MX2050;

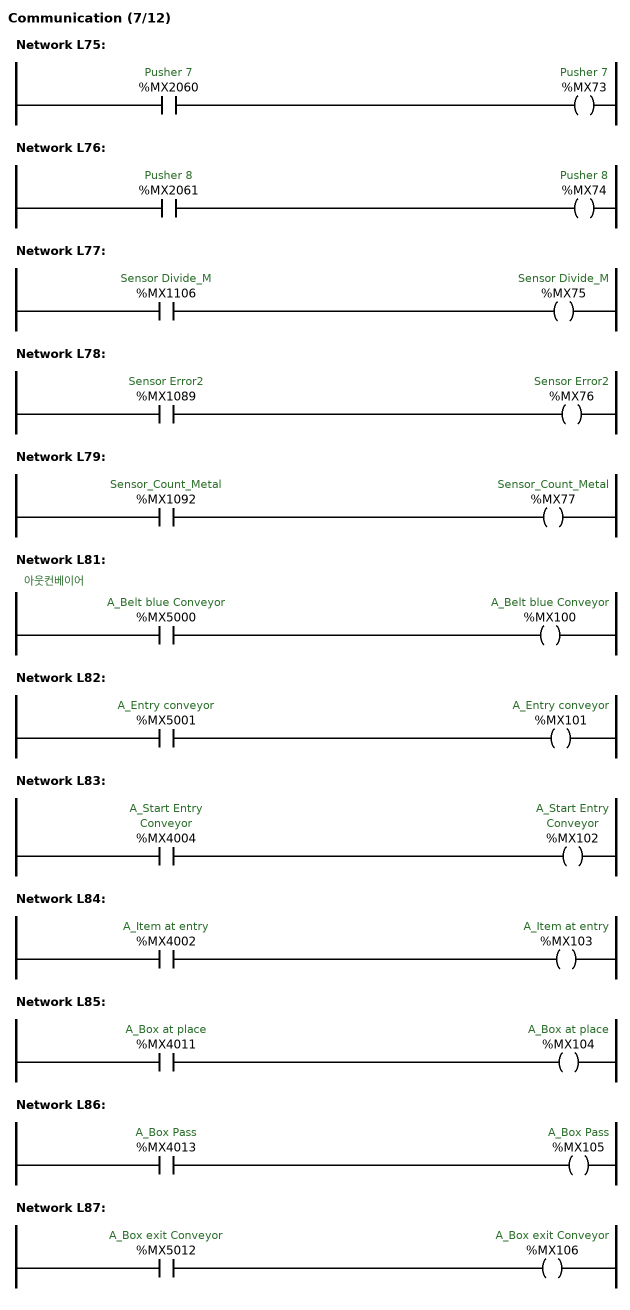
(* Rung L75 *)
%MX73 := %MX2060;
(* Rung L76 *)
%MX74 := %MX2061;
(* Rung L77 *)
%MX75 := %MX1106;
(* Rung L78 *)
%MX76 := %MX1089;
(* Rung L79 *)
%MX77 := %MX1092;
(* 아웃컨베이어 *)
(* Rung L81 *)
%MX100 := %MX5000;
(* Rung L82 *)
%MX101 := %MX5001;
(* Rung L83 *)
%MX102 := %MX4004;
(* Rung L84 *)
%MX103 := %MX4002;
(* Rung L85 *)
%MX104 := %MX4011;
(* Rung L86 *)
%MX105 := %MX4013;
(* Rung L87 *)
%MX106 := %MX5012;

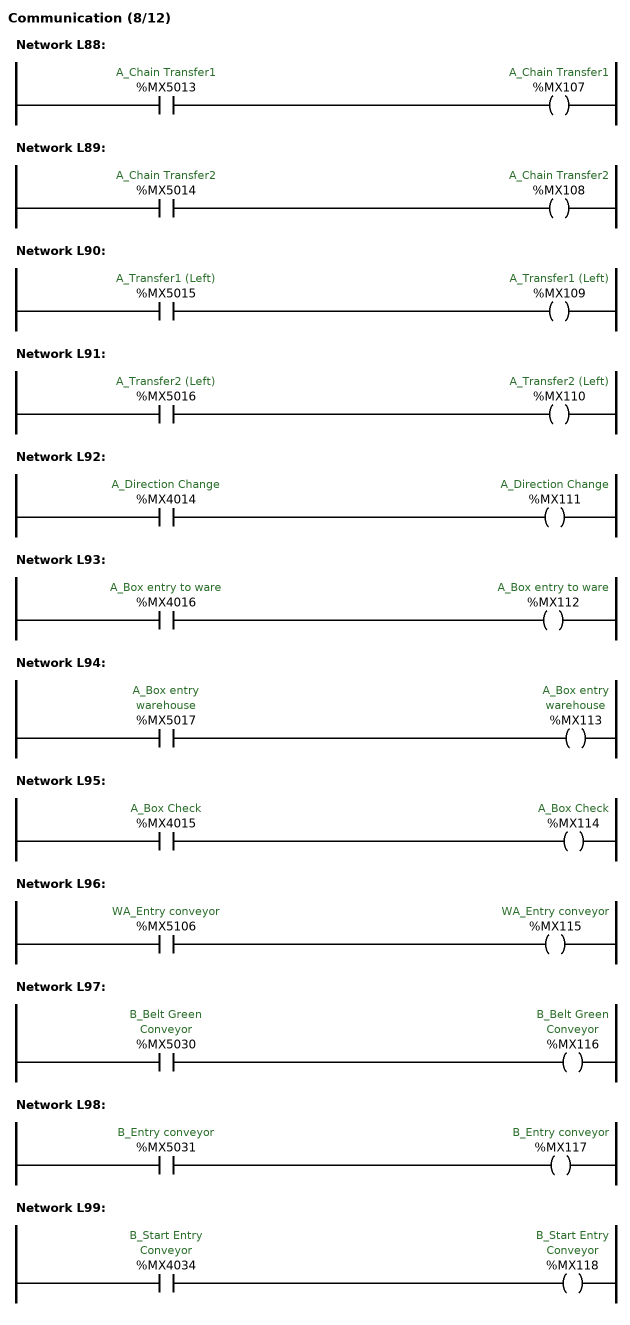
(* Rung L88 *)
%MX107 := %MX5013;
(* Rung L89 *)
%MX108 := %MX5014;
(* Rung L90 *)
%MX109 := %MX5015;
(* Rung L91 *)
%MX110 := %MX5016;
(* Rung L92 *)
%MX111 := %MX4014;
(* Rung L93 *)
%MX112 := %MX4016;
(* Rung L94 *)
%MX113 := %MX5017;
(* Rung L95 *)
%MX114 := %MX4015;
(* Rung L96 *)
%MX115 := %MX5106;
(* Rung L97 *)
%MX116 := %MX5030;
(* Rung L98 *)
%MX117 := %MX5031;
(* Rung L99 *)
%MX118 := %MX4034;

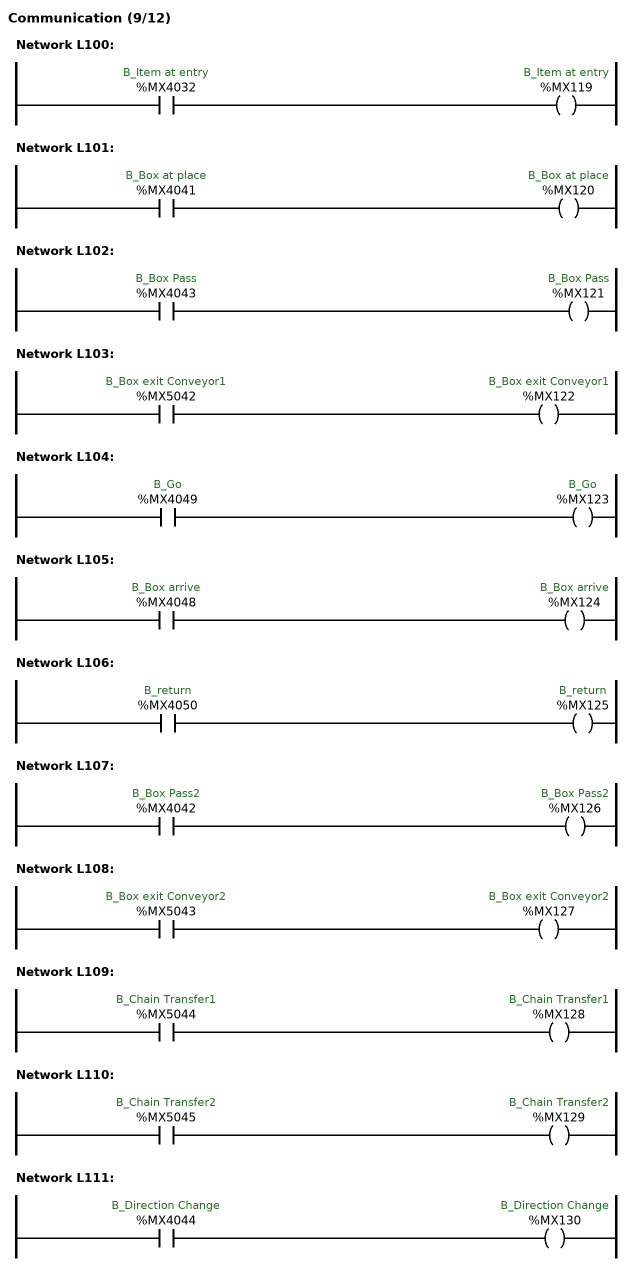
(* Rung L100 *)
%MX119 := %MX4032;
(* Rung L101 *)
%MX120 := %MX4041;
(* Rung L102 *)
%MX121 := %MX4043;
(* Rung L103 *)
%MX122 := %MX5042;
(* Rung L104 *)
%MX123 := %MX4049;
(* Rung L105 *)
%MX124 := %MX4048;
(* Rung L106 *)
%MX125 := %MX4050;
(* Rung L107 *)
%MX126 := %MX4042;
(* Rung L108 *)
%MX127 := %MX5043;
(* Rung L109 *)
%MX128 := %MX5044;
(* Rung L110 *)
%MX129 := %MX5045;
(* Rung L111 *)
%MX130 := %MX4044;

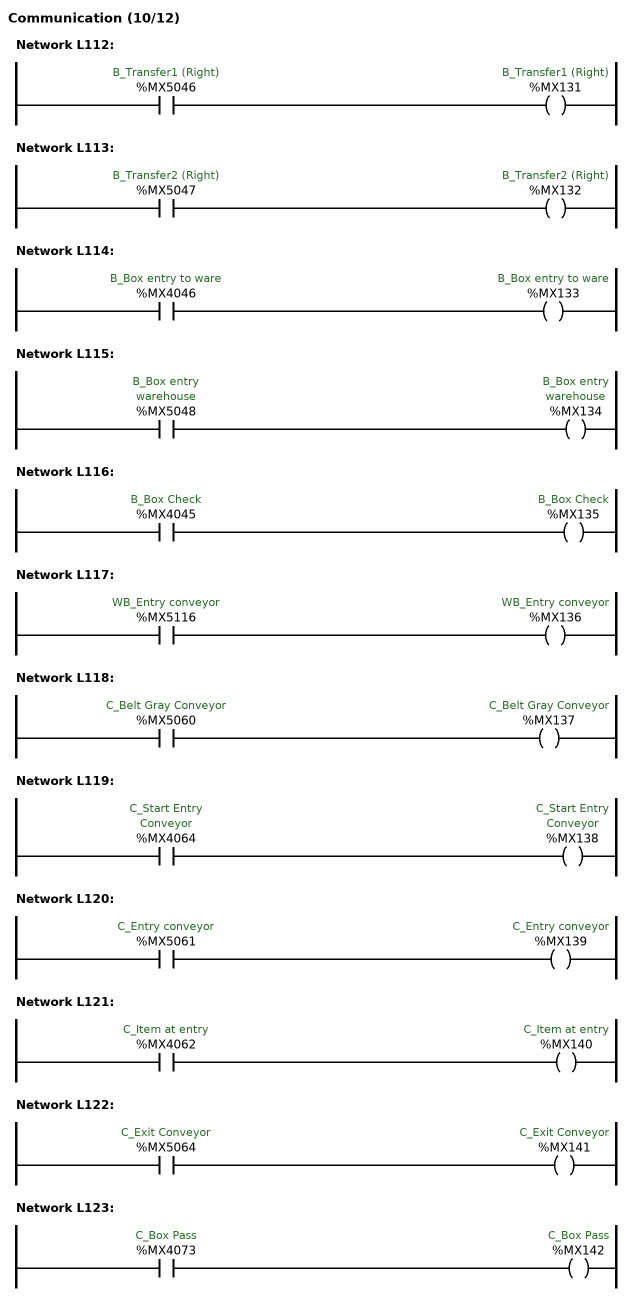
(* Rung L112 *)
%MX131 := %MX5046;
(* Rung L113 *)
%MX132 := %MX5047;
(* Rung L114 *)
%MX133 := %MX4046;
(* Rung L115 *)
%MX134 := %MX5048;
(* Rung L116 *)
%MX135 := %MX4045;
(* Rung L117 *)
%MX136 := %MX5116;
(* Rung L118 *)
%MX137 := %MX5060;
(* Rung L119 *)
%MX138 := %MX4064;
(* Rung L120 *)
%MX139 := %MX5061;
(* Rung L121 *)
%MX140 := %MX4062;
(* Rung L122 *)
%MX141 := %MX5064;
(* Rung L123 *)
%MX142 := %MX4073;

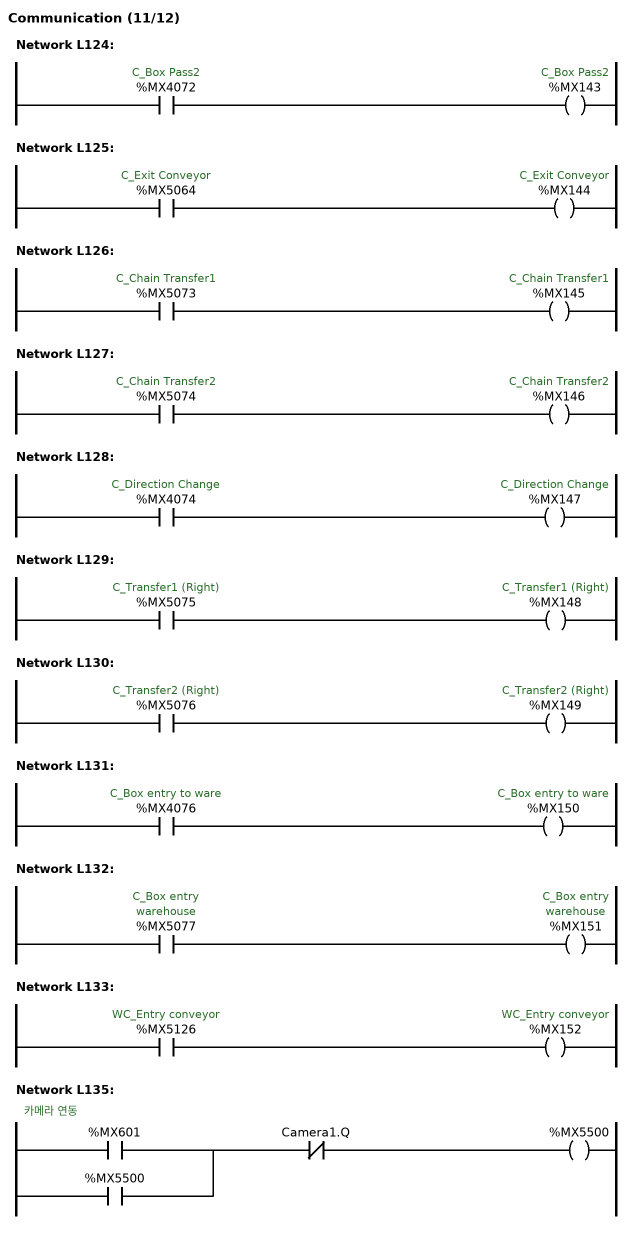
(* Rung L124 *)
%MX143 := %MX4072;
(* Rung L125 *)
%MX144 := %MX5064;
(* Rung L126 *)
%MX145 := %MX5073;
(* Rung L127 *)
%MX146 := %MX5074;
(* Rung L128 *)
%MX147 := %MX4074;
(* Rung L129 *)
%MX148 := %MX5075;
(* Rung L130 *)
%MX149 := %MX5076;
(* Rung L131 *)
%MX150 := %MX4076;
(* Rung L132 *)
%MX151 := %MX5077;
(* Rung L133 *)
%MX152 := %MX5126;
(* 카메라 연동 *)
(* Rung L135 *)
%MX5500 := (%MX601 OR %MX5500) AND NOT Camera1.Q;

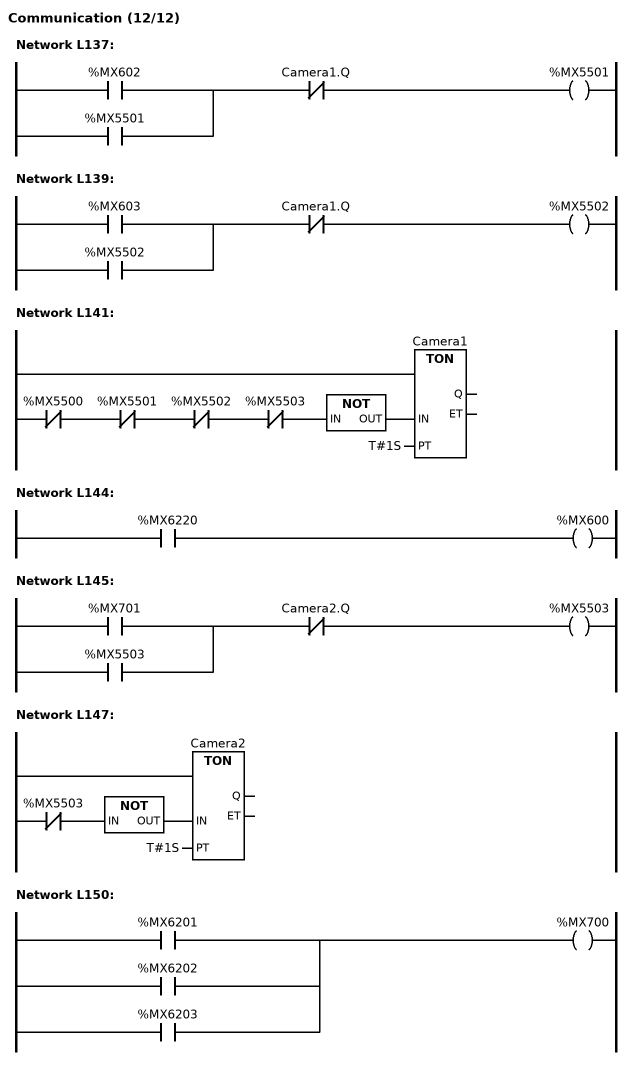
(* Rung L137 *)
%MX5501 := (%MX602 OR %MX5501) AND NOT Camera1.Q;
(* Rung L139 *)
%MX5502 := (%MX603 OR %MX5502) AND NOT Camera1.Q;
(* Rung L141 *)
Camera1(IN := NOT (NOT %MX5500 AND NOT %MX5501 AND NOT %MX5502 AND NOT %MX5503), PT := T#1S);
(* Rung L144 *)
%MX600 := %MX6220;
(* Rung L145 *)
%MX5503 := (%MX701 OR %MX5503) AND NOT Camera2.Q;
(* Rung L147 *)
Camera2(IN := NOT (NOT %MX5503), PT := T#1S);
(* Rung L150 *)
%MX700 := %MX6201 OR %MX6202 OR %MX6203;
END_PROGRAM